{attribute 'qualified_only'}
VAR_GLOBAL CONSTANT
	SUPPORTED_SLOTS : T_SaveSlot := 300;
END_VAR

(* stored: Version 1.1.0.1, ProductVersion 3.1.4019.2
   GVL PARAM_MOTION_SAVEPOINT: Id {17d6d649-9e41-4fac-9f86-04c6437659b4}, ParameterList True *)
